INTERFACE I_UserDefinedDatatype EXTENDS I_Datatype

PROPERTY PUBLIC Identifier : T_MAXSTRING
GET
END_GET
END_PROPERTY

END_INTERFACE

(* stored: Version 1.1.0.1, ProductVersion 3.1.4024.12
   Itf I_UserDefinedDatatype: Id {5c10e49a-8446-0119-0479-1593c1893f3a}
   Property Identifier: Id {04cb09dc-7f72-020d-004f-c29896333291}
   Get Get: Id {dac9de76-7974-0110-2888-8c11522082d9} *)
